INTERFACE I_SuctionCup

PROPERTY bIsSuck : BOOL
GET
END_GET
END_PROPERTY

PROPERTY fThreshold : REAL
GET
END_GET
SET
END_SET
END_PROPERTY

METHOD Release : BOOL
VAR_INPUT
END_VAR
END_METHOD

METHOD Suck : BOOL
VAR_INPUT
END_VAR
END_METHOD

END_INTERFACE

(* stored: Version 1.1.0.1, ProductVersion 3.1.4024.12
   Itf I_SuctionCup: Id {ca6ea579-31cc-4588-8303-73da6b918a03}
   Property bIsSuck: Id {da88f749-8002-4503-8723-15e5b0ba4005}
   Get Get: Id {a9ac35ba-5ff8-4ea6-a52f-25128b1fd8c2}
   Property fThreshold: Id {c9da0623-3275-4ca9-ac42-ccd8ad0a1eb0}
   Get Get: Id {5e7c0797-3aab-473c-8890-69e4ce645fe7}
   Set Set: Id {9943b706-7c14-48af-9854-798ed0377612}
   Method Release: Id {9ea40e11-d82b-40d8-bc6e-685e21c97ec3}
   Method Suck: Id {03461c13-ef78-4c23-8f0d-0236a148a01f} *)
